(* Logix 5000 project; controller Proyecto_Garaje Emulate 5570 rev 33.11; software revision 33.00 *)
// Proyecto de puerta de garaje automatizada

TASK T00_MainTask (continuous, watchdog 500 ms) : P00_MainProgram

MODULES
   Local : Emulate 5570 (ICP 2, rev 33.11)
       : vendor 1 type 0 code 15 (ICP 3, rev 1.1, Output RPI 5 ms)
           Local:3:I.Data[1].0   // Boton Fisico Test Luz entre cerrado
           Local:3:I.Data[1].1   // Boton Fisico Test Luz abierto
           Local:3:I.Data[1].2   // Boton Fisico Test Luz cerrado
           Local:3:I.Data[1].3   // Boton Fisico Test Motor Arriba
           Local:3:I.Data[1].4   // Boton Fisico Test Motor Abajo
           Local:3:I.Data[1].16   // Boton Fisico Subir
           Local:3:I.Data[1].17   // Boton Fisico Bajar
           Local:3:I.Data[1].18   // EMERGENCY STOP FISICO
           Local:3:O.Data[0].0   // Salida Fisica Luz entre Cerrado
           Local:3:O.Data[0].1   // Salida Fisica Luz Abierto
           Local:3:O.Data[0].2   // Salida Fisica Luz Cerrado
           Local:3:O.Data[0].3   // Salida Fisica Motor Arriba
           Local:3:O.Data[0].4   // Salida Fisica Motor Abajo
END_MODULES

VAR_GLOBAL   (* controller tags *)
   CS : BOOL := 1;   // Sensor Puerta Cerrada
   ES : BOOL := 1;   // Paro de emergencia
   LA : BOOL;   // Luz Puerta entre Cerrada
   LC : BOOL := 1;   // Luz Puerta Cerrada
   LO : BOOL;   // Luz Puerta Abierta
   MD : BOOL[32];   // Motor Cerrar Puerta
   MOTOR : TIMER[2] := ([0].PRE := 10000, [1].PRE := 10000);   // Simulacion de Subida y Bajada de Puerta
        [0]   // MOTOR BAJAR
        [1]   // MOTOR ARRIBA
   MU : BOOL[32];   // Motor Abrir Puerta
   OFF : BOOL;
   ON : BOOL;
   OS : BOOL;   // Sensor Puerta Abierta
   PBC : BOOL;   // Boton Cerrar Puerta
   PBO : BOOL;   // Boton Abrir Puerta
   TB : BOOL[32];   // botones Test
        [0]   // Test Inicador Entre cerrado
        [1]   // Boton Test Luz Abierto
        [2]   // Boton Test Luz Abierto
        [3]   // Boton Test Motor Subida
        [4]   // Boton Test Motor Bajada
END_VAR

PROGRAM P00_MainProgram   (* main routine R00_MainRoutine *)

ROUTINE R00_MainRoutine   (* ladder *)
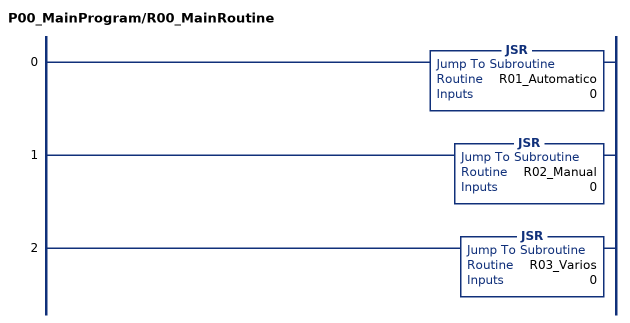
   0: JSR(R01_Automatico,0);
   1: JSR(R02_Manual,0);
   2: JSR(R03_Varios,0);
END_ROUTINE

ROUTINE R01_Automatico   (* ladder *)
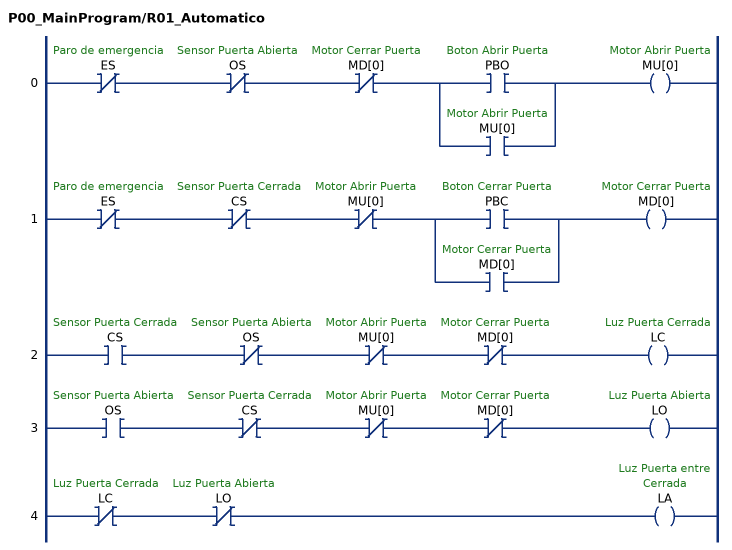
   0: XIO(ES)XIO(OS)XIO(MD[0])[XIC(PBO) ,XIC(MU[0]) ]OTE(MU[0]);
   1: XIO(ES)XIO(CS)XIO(MU[0])[XIC(PBC) ,XIC(MD[0]) ]OTE(MD[0]);
   2: XIC(CS)XIO(OS)XIO(MU[0])XIO(MD[0])OTE(LC);
   3: XIC(OS)XIO(CS)XIO(MU[0])XIO(MD[0])OTE(LO);
   4: XIO(LC)XIO(LO)OTE(LA);
END_ROUTINE

ROUTINE R02_Manual   (* ladder *)
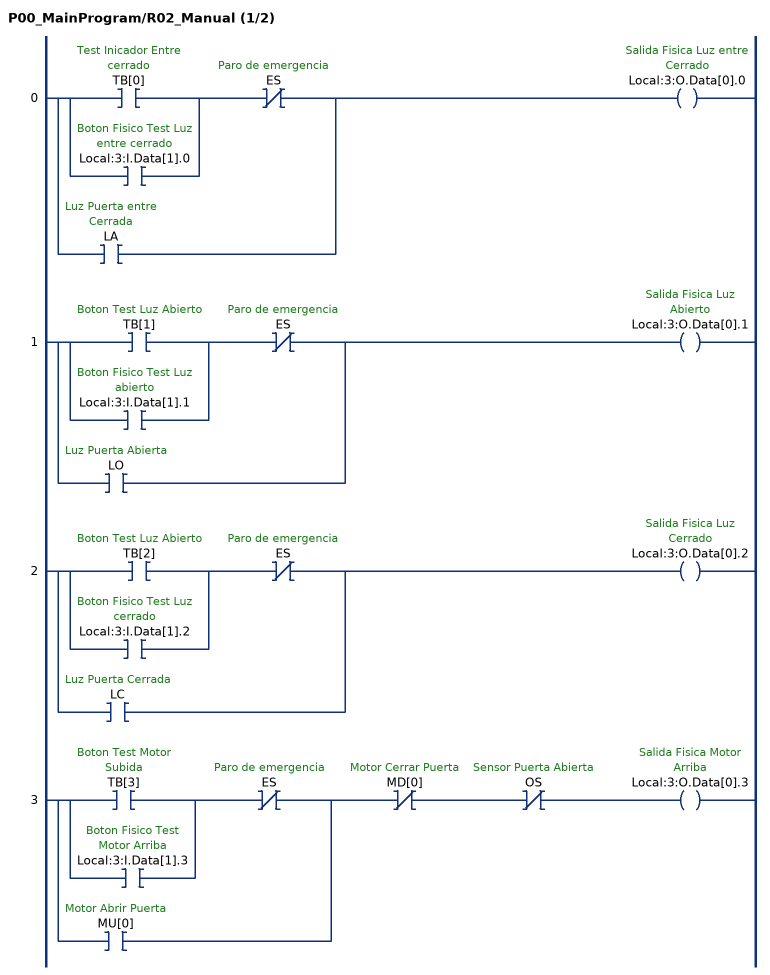
   0: [[XIC(TB[0]) ,XIC(Local:3:I.Data[1].0) ] XIO(ES) ,XIC(LA) ]OTE(Local:3:O.Data[0].0);
   1: [[XIC(TB[1]) ,XIC(Local:3:I.Data[1].1) ] XIO(ES) ,XIC(LO) ]OTE(Local:3:O.Data[0].1);
   2: [[XIC(TB[2]) ,XIC(Local:3:I.Data[1].2) ] XIO(ES) ,XIC(LC) ]OTE(Local:3:O.Data[0].2);
   3: [[XIC(TB[3]) ,XIC(Local:3:I.Data[1].3) ] XIO(ES) ,XIC(MU[0]) ]XIO(MD[0])XIO(OS)OTE(Local:3:O.Data[0].3);
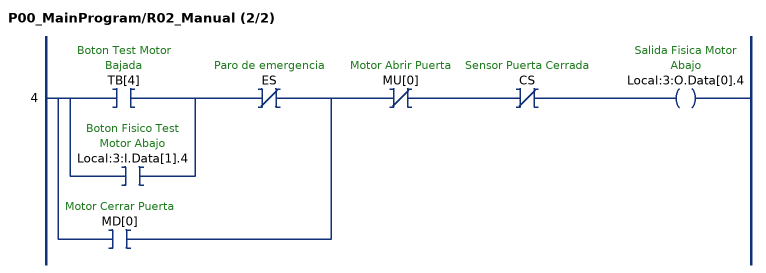
   4: [[XIC(TB[4]) ,XIC(Local:3:I.Data[1].4) ] XIO(ES) ,XIC(MD[0]) ]XIO(MU[0])XIO(CS)OTE(Local:3:O.Data[0].4);
END_ROUTINE

ROUTINE R03_Varios   (* ladder *)
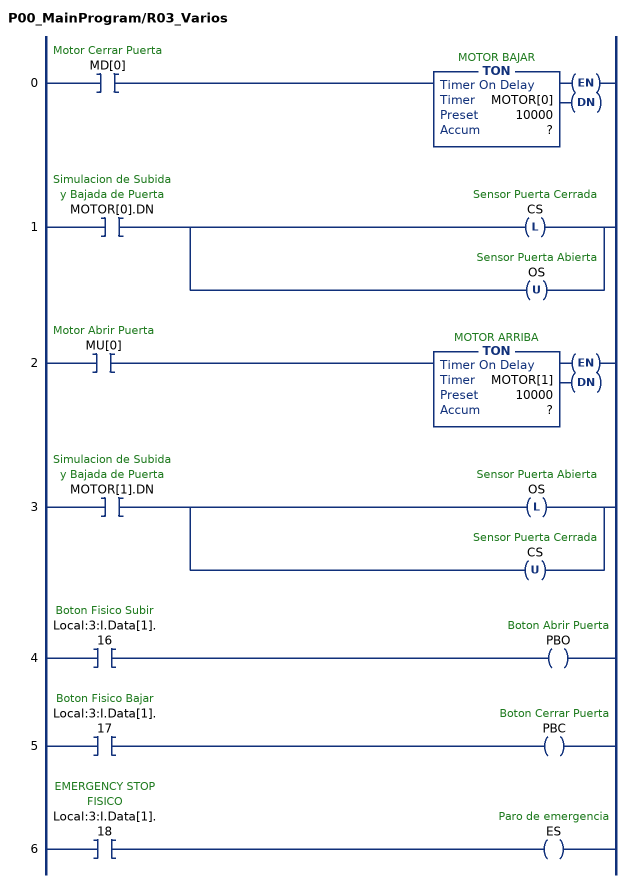
   0: XIC(MD[0])TON(MOTOR[0],?,?);
   1: XIC(MOTOR[0].DN)[OTL(CS) ,OTU(OS) ];
   2: XIC(MU[0])TON(MOTOR[1],?,?);
   3: XIC(MOTOR[1].DN)[OTL(OS) ,OTU(CS) ];
   4: XIC(Local:3:I.Data[1].16)OTE(PBO);
   5: XIC(Local:3:I.Data[1].17)OTE(PBC);
   6: XIC(Local:3:I.Data[1].18)OTE(ES);
END_ROUTINE
END_PROGRAM
